// TIA Portal project "Project10" (V16)

(* hardware
DEVICE "GSD device_1"  GSD.Device.PN
   slot 0: "Rack"  Rack  V1.0
   slot 0: "SINAMICS-V90-PN"  SINAMICS V90 PN V1.0  6SL3 210-5Fxxx-xxFx  V1.00
      slot 0: "SINAMICS V90 PN V1.0"  SINAMICS V90 PN V1.0
      slot 1: "Drive_1"  Drive
         slot 0: "Module Access Point"  Module Access Point
         slot 1: "without PROFIsafe"  without PROFIsafe
      slot 1: "PN-IO"  PN-IO
         slot 1: "Port 1"  Port 1
         slot 2: "Port 2"  Port 2
   slot 2: "Standard telegram 3, PZD-5/9"  Standard telegram 3, PZD-5/9
DEVICE "S7-1200 station_1"  S7-1200 Station
   slot 0: "Rack_0"  S7-1200 Rack  Rack  V1.0
   slot 1: "PLC_1"  CPU 1214C AC/DC/Rly  6ES7 214-1BG40-0XB0  V4.3
*)

// ===== PLC "PLC_1"  CPU 1214C AC/DC/Rly =====

VAR_GLOBAL   // PLC tag table "Default tag table"
   "System_Byte" AT %MB1 : Byte;
   "FirstScan" AT %M1.0 : Bool;
   "DiagStatusUpdate" AT %M1.1 : Bool;
   "AlwaysTRUE" AT %M1.2 : Bool;
   "AlwaysFALSE" AT %M1.3 : Bool;
   "piston_ileri" AT %Q0.0 : Bool;
   "piston_geri" AT %Q0.1 : Bool;
   "pisron1_ilerde_sensörü" AT %I0.0 : Bool;
   "pisron1_geride_sensörü" AT %I0.1 : Bool;
   "pisron2_ilerde_sensörü" AT %I0.2 : Bool;
   "pisron2_geride_sensörü" AT %I0.3 : Bool;
   "hava_var_sinyal" AT %I0.7 : Bool;
   "acil_durum_basılı" AT %I0.4 : Bool;
   "otomatik_röle" AT %M2.0 : Bool;
   "manuel_röle" AT %M2.1 : Bool;
   "manuel_servo" AT %M2.2 : Bool;
   "manuel_piston" AT %M2.3 : Bool;
   "otomatik_hız1" AT %M2.4 : Bool;
   "otomatik_hız2" AT %M2.5 : Bool;
   "manuel_pistonlar_geri" AT %M2.6 : Bool;
   "manuel_pistonlar_ileri" AT %M2.7 : Bool;
   "oto_konum_1" AT %M3.0 : Bool;
   "oto_konum_2" AT %M3.1 : Bool;
   "oto_konum_3" AT %M3.2 : Bool;
   "oto_konum_4" AT %M3.3 : Bool;
   "oto_start" AT %M3.4 : Bool;
   "hız_bilgisi" AT %MD400 : Real;
   "konum_bilgisi" AT %MD450 : Real;
   "servo_on" AT %M12.0 : Bool;
   "servo_reset" AT %M12.1 : Bool;
   "pozisyon_start" AT %M12.2 : Bool;
   "pozisyon_tamamlandı" AT %M12.3 : Bool;
   "home_start" AT %M12.4 : Bool;
   "home_tamamlandı" AT %M12.5 : Bool;
   "Axis_1_Drive_IN" AT %I68.0 : "PD_TEL3_IN";
   "Axis_1_Drive_OUT" AT %Q64.0 : "PD_TEL3_OUT";
   "home_okey" AT %M12.6 : Bool;
   "pozi_okey" AT %M12.7 : Bool;
   "manuel_motor_ileri" AT %M13.0 : Bool;
   "manuel_motor_geri" AT %M13.1 : Bool;
   "oto_piston_ileri_start1" AT %M13.2 : Bool;
   "oto_piston_ileri_start2" AT %M13.3 : Bool;
   "oto_piston_ileri_start3" AT %M13.4 : Bool;
   "oto_piston_ileri_start4" AT %M13.5 : Bool;
   "oto_piston_geri_start1" AT %M13.6 : Bool;
   "oto_piston_geri_start2" AT %M13.7 : Bool;
   "oto_piston_geri_start3" AT %M14.0 : Bool;
   "oto_piston_geri_start4" AT %M14.1 : Bool;
   "sıra_izleme" AT %MW430 : Word;
   "oto_poz_start1" AT %M14.2 : Bool;
   "oto_poz_start2" AT %M14.3 : Bool;
   "oto_poz_start3" AT %M14.4 : Bool;
   "oto_poz_start4" AT %M14.5 : Bool;
   "oto_poz_start5" AT %M14.6 : Bool;
   "Tag_1" AT %M99.1 : Bool;
   "poz_set_düşür1" AT %M99.2 : Bool;
   "poz_set_düşür2" AT %M99.3 : Bool;
   "poz_set_düşür3" AT %M99.4 : Bool;
   "poz_set_düşür4" AT %M99.5 : Bool;
   "timer_set" AT %M99.6 : Bool;
   "Tag_2" AT %M98.0 : Bool;
   "timer_reset" AT %M98.1 : Bool;
   "servo_busy" AT %M98.2 : Bool;
   "hız1" AT %MD100 : Real;
   "arttırma" AT %M98.3 : Bool;
   "jog_meşgul" AT %M98.4 : Bool;
   "deneme" AT %M98.5 : Bool;
   "Clock_Byte" AT %MB0 : Byte;
   "Clock_10Hz" AT %M0.0 : Bool;
   "Clock_5Hz" AT %M0.1 : Bool;
   "Clock_2.5Hz" AT %M0.2 : Bool;
   "Clock_2Hz" AT %M0.3 : Bool;
   "Clock_1.25Hz" AT %M0.4 : Bool;
   "Clock_1Hz" AT %M0.5 : Bool;
   "Clock_0.625Hz" AT %M0.6 : Bool;
   "Clock_0.5Hz" AT %M0.7 : Bool;
   "COU_RST" AT %M3.5 : Bool;
   "DEN" AT %M3.6 : Bool;
END_VAR

DATA_BLOCK "DB_QR_DENEME"   // DB2
{ S7_Optimized_Access := 'FALSE' }
VERSION : 0.1
   VAR
      otomatik_manuel_mod_seçimi : Bool;
      manuel_seçim1 : Bool;
      manuel_seçim2 : Bool;
      manuel_piston_durum_oto_hız_bilgisi_1 : Bool;
      manuel_piston_durum_oto_hız_bilgisi_2 : Bool;
      oto_konum_bilgisi_1 : Bool;
      oto_konum_bilgisi_2 : Bool;
      oto_start : Bool;
      hız : Real;
      konum : Real;
      konum2 : Real;
      manuel_karşılaştır : Bool;
      sin : Bool;
      sinyal_oku2 : Bool;
      sinyal_oku : Bool;
   END_VAR
BEGIN
END_DATA_BLOCK

DATA_BLOCK "dbGenel"   // DB11
{ S7_Optimized_Access := 'TRUE' }
VERSION : 0.1
   VAR
      count : IEC_UCOUNTER;
   END_VAR
   VAR RETAIN
      Mikta : UInt;
   END_VAR
   VAR
      P_ken : Array[0..10] of Bool;
      reset : Bool;
      deneme : Bool;
      deneme_1 : Bool;
      deneme_2 : Bool;
   END_VAR
BEGIN
END_DATA_BLOCK

// folder: System blocks/Program resources

DATA_BLOCK "IEC_Timer_0_DB"   // DB8
{ S7_Optimized_Access := 'TRUE' }
AUTHOR : Simatic
FAMILY : IEC
NAME : IEC_TMR
VERSION : 1.0
// stored: InstanceOfName IEC_TIMER
"IEC_TIMER"
BEGIN
END_DATA_BLOCK

DATA_BLOCK "IEC_Timer_0_DB_1"   // DB9
{ S7_Optimized_Access := 'TRUE' }
AUTHOR : Simatic
FAMILY : IEC
NAME : IEC_TMR
VERSION : 1.0
// stored: InstanceOfName IEC_TIMER
"IEC_TIMER"
BEGIN
END_DATA_BLOCK

DATA_BLOCK "IEC_Timer_0_DB_2"   // DB10
{ S7_Optimized_Access := 'TRUE' }
AUTHOR : Simatic
FAMILY : IEC
NAME : IEC_TMR
VERSION : 1.0
// stored: InstanceOfName IEC_TIMER
"IEC_TIMER"
BEGIN
END_DATA_BLOCK

DATA_BLOCK "IEC_Timer_0_DB_5"   // DB13
{ S7_Optimized_Access := 'TRUE' }
AUTHOR : Simatic
FAMILY : IEC
NAME : IEC_TMR
VERSION : 1.0
// stored: InstanceOfName IEC_TIMER
"IEC_TIMER"
BEGIN
END_DATA_BLOCK

DATA_BLOCK "IEC_Counter_0_DB_1"   // DB14
{ S7_Optimized_Access := 'TRUE' }
AUTHOR : Simatic
FAMILY : IEC
NAME : CNTR
VERSION : 1.0
// stored: InstanceOfName IEC_COUNTER
"IEC_COUNTER"
BEGIN
END_DATA_BLOCK

// folder: (top level)

DATA_BLOCK "Axis_1"   // DB1, Motion_DB
{ S7_Optimized_Access := 'TRUE' }
AUTHOR : SIMATIC
FAMILY : BasicMC
NAME : TO_PosAx
VERSION : 6.0
// stored: InstanceOfName TO_PositioningAxis
"TO_PositioningAxis"
BEGIN
   // Axis.Encoder.TelegramAddressOutCU = %Q64.0
   // Axis.Encoder.TelegramAddressInCU = %I68.0
   // Axis.Encoder.DoNameCU = SINAMICS-V90-PN.Drive_1_Encoder1
   // Axis.Drive.TelegramAddressOutCU = %Q64.0
   // Axis.Drive.TelegramAddressInCU = %I68.0
   // Axis.Drive.TelegramType = 2
   // Axis.Drive.DoNameCU = SINAMICS-V90-PN.Drive_1
   // Axis.LengthUnitNormalized.Time = 1
   // Axis.LengthUnitNormalized.Distance = -2
   // Axis.Encoder.SelectedHscIndexCU = -1
   // Axis.Encoder.DbTypeCU = Classic
   // Axis.Drive.DbTypeCU = Classic
END_DATA_BLOCK

FUNCTION "fc_qr_eşleştir" : Void   // FC1, LAD
{ S7_Optimized_Access := 'TRUE' }
VERSION : 0.1
   VAR_TEMP   // added for the SCL form of the ladder/FBD networks
      _w1 : Bool;
   END_VAR
BEGIN

REGION Network 1: otomatik_manuel_mod_seçimi
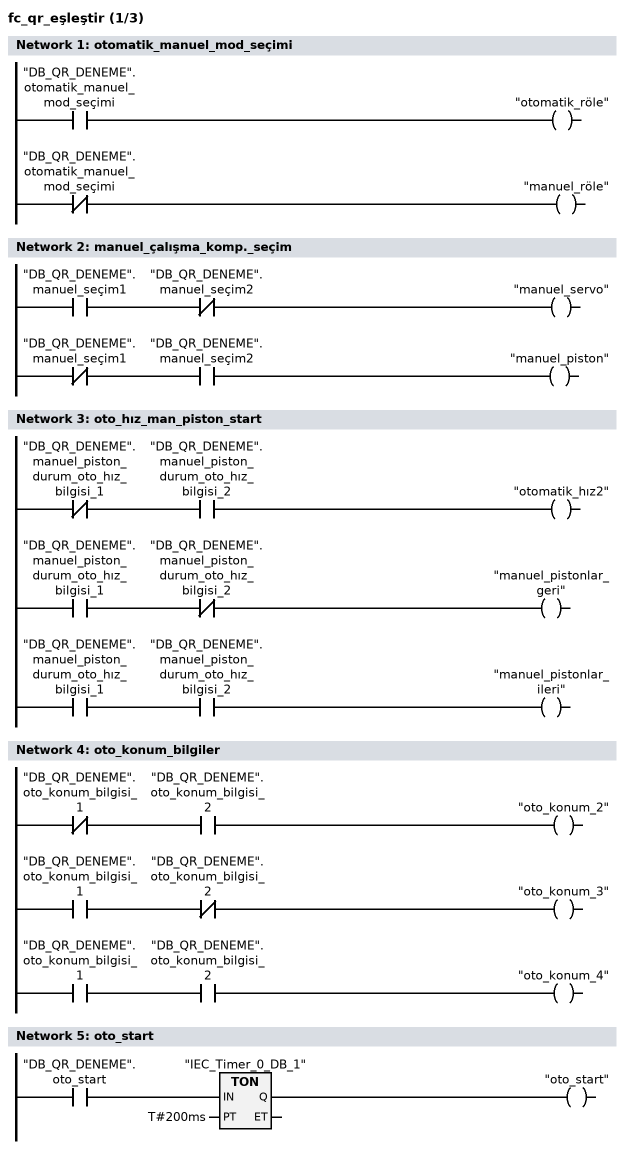
   RUNG wire#powerrail
      Contact( "DB_QR_DENEME".otomatik_manuel_mod_seçimi )
      Coil( "otomatik_röle" )
   END_RUNG
   RUNG wire#powerrail
      I_Contact( "DB_QR_DENEME".otomatik_manuel_mod_seçimi )
      Coil( "manuel_röle" )
   END_RUNG
   // the same network as SCL:
   "otomatik_röle" := "DB_QR_DENEME".otomatik_manuel_mod_seçimi;
   "manuel_röle" := NOT "DB_QR_DENEME".otomatik_manuel_mod_seçimi;
END_REGION

REGION Network 2: manuel_çalışma_komp._seçim
   RUNG wire#powerrail
      Contact( "DB_QR_DENEME".manuel_seçim1 )
      I_Contact( "DB_QR_DENEME".manuel_seçim2 )
      Coil( "manuel_servo" )
   END_RUNG
   RUNG wire#powerrail
      I_Contact( "DB_QR_DENEME".manuel_seçim1 )
      Contact( "DB_QR_DENEME".manuel_seçim2 )
      Coil( "manuel_piston" )
   END_RUNG
   // the same network as SCL:
   "manuel_servo" := "DB_QR_DENEME".manuel_seçim1 AND NOT "DB_QR_DENEME".manuel_seçim2;
   "manuel_piston" := NOT "DB_QR_DENEME".manuel_seçim1 AND "DB_QR_DENEME".manuel_seçim2;
END_REGION

REGION Network 3: oto_hız_man_piston_start
   RUNG wire#powerrail
      I_Contact( "DB_QR_DENEME".manuel_piston_durum_oto_hız_bilgisi_1 )
      Contact( "DB_QR_DENEME".manuel_piston_durum_oto_hız_bilgisi_2 )
      Coil( "otomatik_hız2" )
   END_RUNG
   RUNG wire#powerrail
      Contact( "DB_QR_DENEME".manuel_piston_durum_oto_hız_bilgisi_1 )
      I_Contact( "DB_QR_DENEME".manuel_piston_durum_oto_hız_bilgisi_2 )
      Coil( "manuel_pistonlar_geri" )
   END_RUNG
   RUNG wire#powerrail
      Contact( "DB_QR_DENEME".manuel_piston_durum_oto_hız_bilgisi_1 )
      Contact( "DB_QR_DENEME".manuel_piston_durum_oto_hız_bilgisi_2 )
      Coil( "manuel_pistonlar_ileri" )
   END_RUNG
   // the same network as SCL:
   "otomatik_hız2" := NOT "DB_QR_DENEME".manuel_piston_durum_oto_hız_bilgisi_1 AND "DB_QR_DENEME".manuel_piston_durum_oto_hız_bilgisi_2;
   "manuel_pistonlar_geri" := "DB_QR_DENEME".manuel_piston_durum_oto_hız_bilgisi_1 AND NOT "DB_QR_DENEME".manuel_piston_durum_oto_hız_bilgisi_2;
   "manuel_pistonlar_ileri" := "DB_QR_DENEME".manuel_piston_durum_oto_hız_bilgisi_1 AND "DB_QR_DENEME".manuel_piston_durum_oto_hız_bilgisi_2;
END_REGION

REGION Network 4: oto_konum_bilgiler
   RUNG wire#powerrail
      I_Contact( "DB_QR_DENEME".oto_konum_bilgisi_1 )
      Contact( "DB_QR_DENEME".oto_konum_bilgisi_2 )
      Coil( "oto_konum_2" )
   END_RUNG
   RUNG wire#powerrail
      Contact( "DB_QR_DENEME".oto_konum_bilgisi_1 )
      I_Contact( "DB_QR_DENEME".oto_konum_bilgisi_2 )
      Coil( "oto_konum_3" )
   END_RUNG
   RUNG wire#powerrail
      Contact( "DB_QR_DENEME".oto_konum_bilgisi_1 )
      Contact( "DB_QR_DENEME".oto_konum_bilgisi_2 )
      Coil( "oto_konum_4" )
   END_RUNG
   // the same network as SCL:
   "oto_konum_2" := NOT "DB_QR_DENEME".oto_konum_bilgisi_1 AND "DB_QR_DENEME".oto_konum_bilgisi_2;
   "oto_konum_3" := "DB_QR_DENEME".oto_konum_bilgisi_1 AND NOT "DB_QR_DENEME".oto_konum_bilgisi_2;
   "oto_konum_4" := "DB_QR_DENEME".oto_konum_bilgisi_1 AND "DB_QR_DENEME".oto_konum_bilgisi_2;
END_REGION

REGION Network 5: oto_start
   "IEC_Timer_0_DB_1".TON(IN := "DB_QR_DENEME".oto_start, PT := T#200ms);
   "oto_start" := "IEC_Timer_0_DB_1".Q;
END_REGION

REGION Network 6: hız_konum_atama
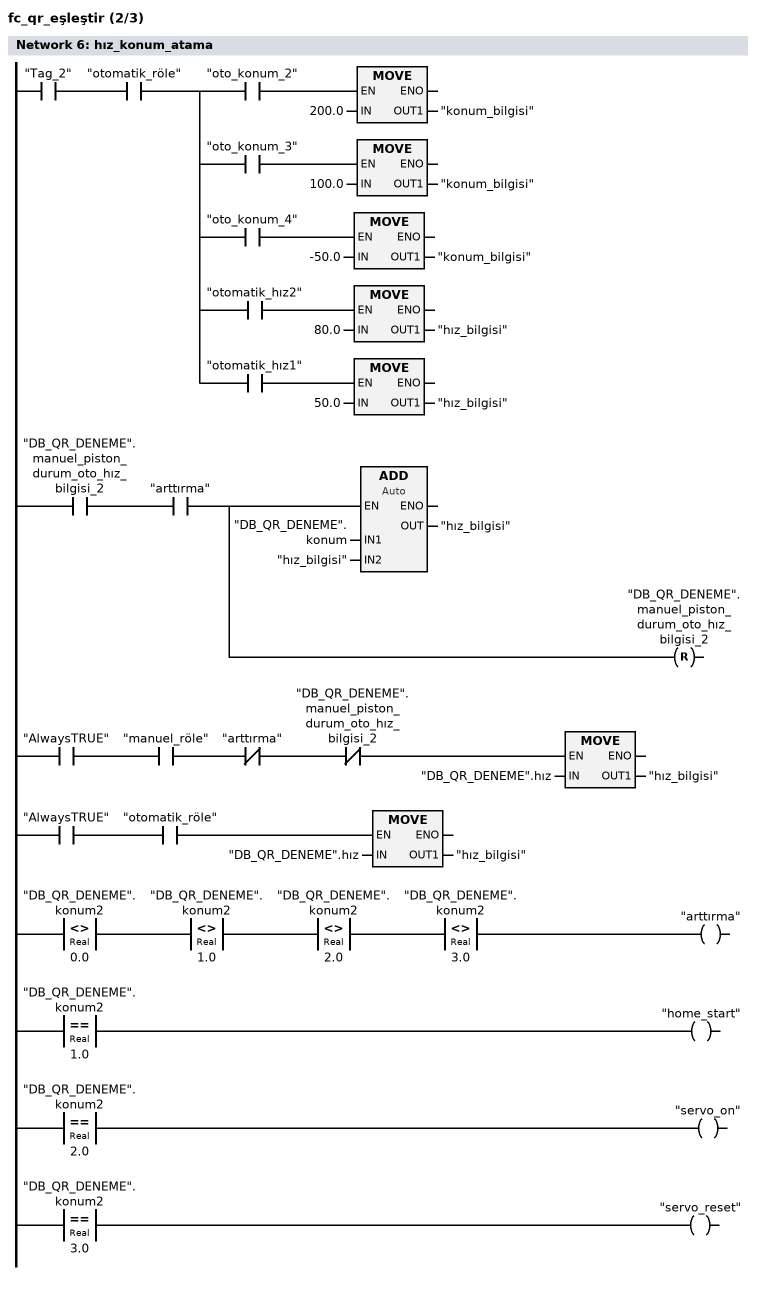
   RUNG wire#powerrail
      Contact( "Tag_2" )
      Contact( "otomatik_röle" )
      wire#w1
      Contact( "oto_konum_2" )
      Move(in := 200.0, out1 => "konum_bilgisi")
   END_RUNG
   RUNG wire#w1
      Contact( "oto_konum_3" )
      Move(in := 100.0, out1 => "konum_bilgisi")
   END_RUNG
   RUNG wire#w1
      Contact( "oto_konum_4" )
      Move(in := -50.0, out1 => "konum_bilgisi")
   END_RUNG
   RUNG wire#w1
      Contact( "otomatik_hız2" )
      Move(in := 80.0, out1 => "hız_bilgisi")
   END_RUNG
   RUNG wire#w1
      Contact( "otomatik_hız1" )
      Move(in := 50.0, out1 => "hız_bilgisi")
   END_RUNG
   RUNG wire#powerrail
      Contact( "DB_QR_DENEME".manuel_piston_durum_oto_hız_bilgisi_2 )
      Contact( "arttırma" )
      wire#w2
      Add(in1 := "DB_QR_DENEME".konum, in2 := "hız_bilgisi", out => "hız_bilgisi")
   END_RUNG
   RUNG wire#w2
      R_Coil( "DB_QR_DENEME".manuel_piston_durum_oto_hız_bilgisi_2 )
   END_RUNG
   RUNG wire#powerrail
      Contact( "AlwaysTRUE" )
      Contact( "manuel_röle" )
      I_Contact( "arttırma" )
      I_Contact( "DB_QR_DENEME".manuel_piston_durum_oto_hız_bilgisi_2 )
      Move(in := "DB_QR_DENEME".hız, out1 => "hız_bilgisi")
   END_RUNG
   RUNG wire#powerrail
      Contact( "AlwaysTRUE" )
      Contact( "otomatik_röle" )
      Move(in := "DB_QR_DENEME".hız, out1 => "hız_bilgisi")
   END_RUNG
   RUNG wire#powerrail
      { S7_Templates := "SrcType := Real" } NE_Contact(in1 := "DB_QR_DENEME".konum2, in2 := 0.0)
      { S7_Templates := "SrcType := Real" } NE_Contact(in1 := "DB_QR_DENEME".konum2, in2 := 1.0)
      { S7_Templates := "SrcType := Real" } NE_Contact(in1 := "DB_QR_DENEME".konum2, in2 := 2.0)
      { S7_Templates := "SrcType := Real" } NE_Contact(in1 := "DB_QR_DENEME".konum2, in2 := 3.0)
      Coil( "arttırma" )
   END_RUNG
   RUNG wire#powerrail
      { S7_Templates := "SrcType := Real" } EQ_Contact(in1 := "DB_QR_DENEME".konum2, in2 := 1.0)
      Coil( "home_start" )
   END_RUNG
   RUNG wire#powerrail
      { S7_Templates := "SrcType := Real" } EQ_Contact(in1 := "DB_QR_DENEME".konum2, in2 := 2.0)
      Coil( "servo_on" )
   END_RUNG
   RUNG wire#powerrail
      { S7_Templates := "SrcType := Real" } EQ_Contact(in1 := "DB_QR_DENEME".konum2, in2 := 3.0)
      Coil( "servo_reset" )
   END_RUNG
   // the same network as SCL:
   #_w1 := "Tag_2" AND "otomatik_röle";
   IF #_w1 AND "oto_konum_2" THEN "konum_bilgisi" := 200.0; END_IF;
   IF #_w1 AND "oto_konum_3" THEN "konum_bilgisi" := 100.0; END_IF;
   IF #_w1 AND "oto_konum_4" THEN "konum_bilgisi" := -50.0; END_IF;
   IF #_w1 AND "otomatik_hız2" THEN "hız_bilgisi" := 80.0; END_IF;
   IF #_w1 AND "otomatik_hız1" THEN "hız_bilgisi" := 50.0; END_IF;
   IF "DB_QR_DENEME".manuel_piston_durum_oto_hız_bilgisi_2 AND "arttırma" THEN
       "hız_bilgisi" := "DB_QR_DENEME".konum + "hız_bilgisi";
       "DB_QR_DENEME".manuel_piston_durum_oto_hız_bilgisi_2 := FALSE;
   END_IF;
   IF "AlwaysTRUE" AND "manuel_röle" AND NOT "arttırma" AND NOT "DB_QR_DENEME".manuel_piston_durum_oto_hız_bilgisi_2 THEN
       "hız_bilgisi" := "DB_QR_DENEME".hız;
   END_IF;
   IF "AlwaysTRUE" AND "otomatik_röle" THEN "hız_bilgisi" := "DB_QR_DENEME".hız; END_IF;
   "arttırma" := ("DB_QR_DENEME".konum2 <> 0.0) AND ("DB_QR_DENEME".konum2 <> 1.0) AND ("DB_QR_DENEME".konum2 <> 2.0) AND ("DB_QR_DENEME".konum2 <> 3.0);
   "home_start" := "DB_QR_DENEME".konum2 = 1.0;
   "servo_on" := "DB_QR_DENEME".konum2 = 2.0;
   "servo_reset" := "DB_QR_DENEME".konum2 = 3.0;
END_REGION

REGION Network 7
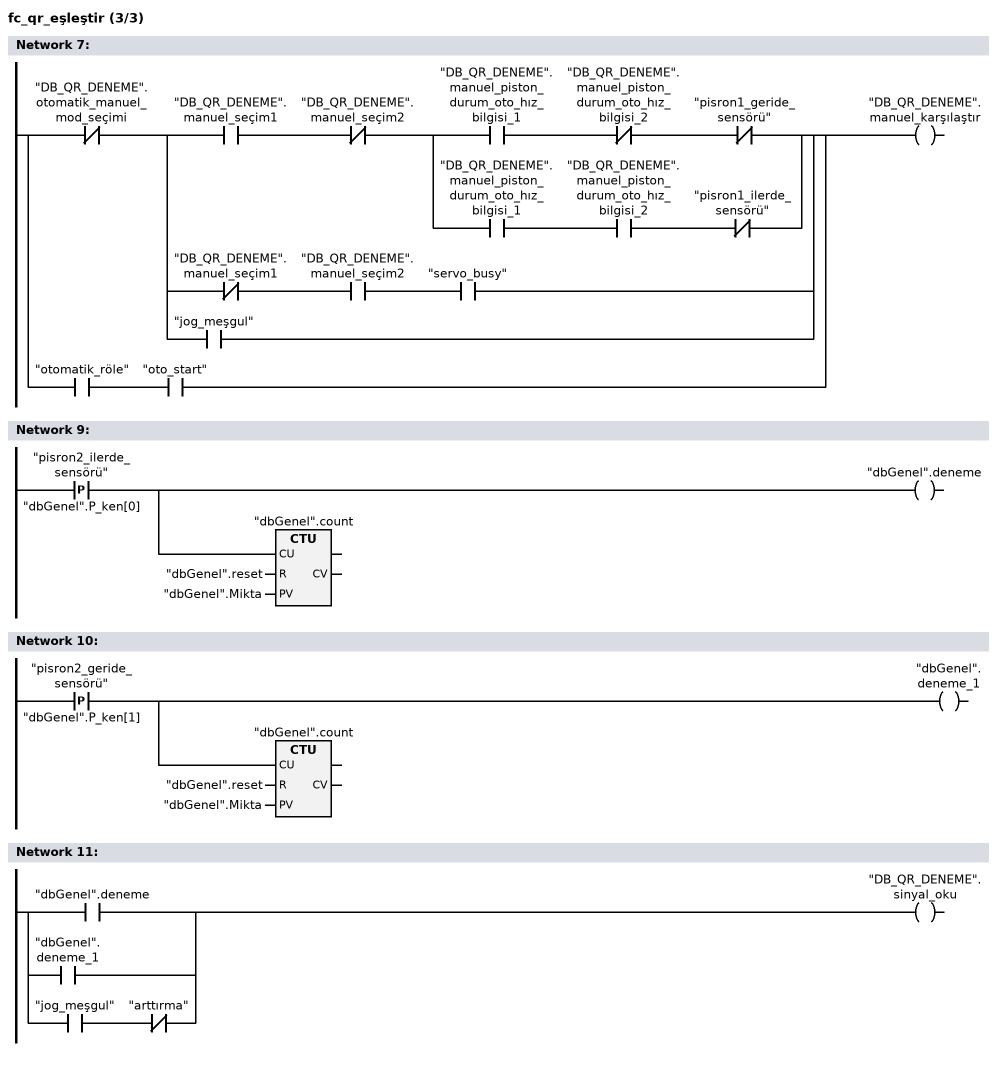
   RUNG wire#powerrail
      I_Contact( "DB_QR_DENEME".otomatik_manuel_mod_seçimi )
      wire#w1
      Contact( "DB_QR_DENEME".manuel_seçim1 )
      I_Contact( "DB_QR_DENEME".manuel_seçim2 )
      wire#w2
      Contact( "DB_QR_DENEME".manuel_piston_durum_oto_hız_bilgisi_1 )
      I_Contact( "DB_QR_DENEME".manuel_piston_durum_oto_hız_bilgisi_2 )
      I_Contact( "pisron1_geride_sensörü" )
      wire#w3
      Coil( "DB_QR_DENEME".manuel_karşılaştır )
   END_RUNG
   RUNG wire#w2
      Contact( "DB_QR_DENEME".manuel_piston_durum_oto_hız_bilgisi_1 )
      Contact( "DB_QR_DENEME".manuel_piston_durum_oto_hız_bilgisi_2 )
      I_Contact( "pisron1_ilerde_sensörü" )
   END_RUNG wire#w3
   RUNG wire#w1
      I_Contact( "DB_QR_DENEME".manuel_seçim1 )
      Contact( "DB_QR_DENEME".manuel_seçim2 )
      Contact( "servo_busy" )
   END_RUNG wire#w3
   RUNG wire#w1
      Contact( "jog_meşgul" )
   END_RUNG wire#w3
   RUNG wire#powerrail
      Contact( "otomatik_röle" )
      Contact( "oto_start" )
   END_RUNG wire#w3
   // the same network as SCL:
   "DB_QR_DENEME".manuel_karşılaştır := (NOT "DB_QR_DENEME".otomatik_manuel_mod_seçimi AND (("DB_QR_DENEME".manuel_seçim1 AND NOT "DB_QR_DENEME".manuel_seçim2 AND (("DB_QR_DENEME".manuel_piston_durum_oto_hız_bilgisi_1 AND NOT "DB_QR_DENEME".manuel_piston_durum_oto_hız_bilgisi_2 AND NOT "pisron1_geride_sensörü") OR ("DB_QR_DENEME".manuel_piston_durum_oto_hız_bilgisi_1 AND "DB_QR_DENEME".manuel_piston_durum_oto_hız_bilgisi_2 AND NOT "pisron1_ilerde_sensörü"))) OR (NOT "DB_QR_DENEME".manuel_seçim1 AND "DB_QR_DENEME".manuel_seçim2 AND "servo_busy") OR "jog_meşgul")) OR ("otomatik_röle" AND "oto_start");
END_REGION

REGION Network 9
   #_w1 := "pisron2_ilerde_sensörü" AND NOT "dbGenel".P_ken[0];   // rising edge of "pisron2_ilerde_sensörü"
   "dbGenel".P_ken[0] := "pisron2_ilerde_sensörü";
   "dbGenel".deneme := #_w1;
   "dbGenel".count.CTU(CU := #_w1, R := "dbGenel".reset, PV := "dbGenel".Mikta);
END_REGION

REGION Network 10
   #_w1 := "pisron2_geride_sensörü" AND NOT "dbGenel".P_ken[1];   // rising edge of "pisron2_geride_sensörü"
   "dbGenel".P_ken[1] := "pisron2_geride_sensörü";
   "dbGenel".deneme_1 := #_w1;
   "dbGenel".count.CTU(CU := #_w1, R := "dbGenel".reset, PV := "dbGenel".Mikta);
END_REGION

REGION Network 11
   RUNG wire#powerrail
      Contact( "dbGenel".deneme )
      wire#w1
      Coil( "DB_QR_DENEME".sinyal_oku )
   END_RUNG
   RUNG wire#powerrail
      Contact( "dbGenel".deneme_1 )
   END_RUNG wire#w1
   RUNG wire#powerrail
      Contact( "jog_meşgul" )
      I_Contact( "arttırma" )
   END_RUNG wire#w1
   // the same network as SCL:
   "DB_QR_DENEME".sinyal_oku := "dbGenel".deneme OR "dbGenel".deneme_1 OR ("jog_meşgul" AND NOT "arttırma");
END_REGION
END_FUNCTION

FUNCTION "fc_servo" : Void   // FC2, LAD
{ S7_Optimized_Access := 'TRUE' }
VERSION : 0.1
BEGIN

REGION Network 1
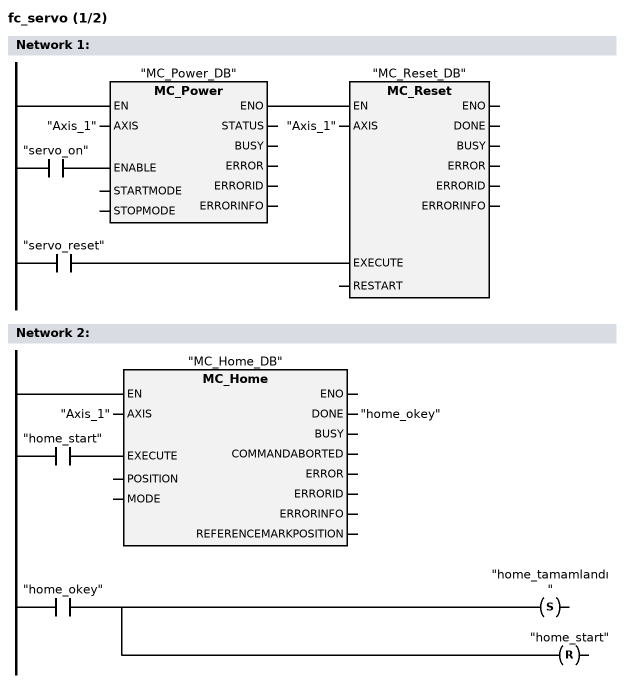
   // ENO of a box is taken as its EN; it also drops when the box reports an error
   "MC_Power_DB"(Axis := "Axis_1", Enable := "servo_on");   // MC_Power
   "MC_Reset_DB"(Axis := "Axis_1", Execute := "servo_reset");   // MC_Reset
END_REGION

REGION Network 2
   "MC_Home_DB"(Axis := "Axis_1", Execute := "home_start", Done => "home_okey");   // MC_Home
   IF "home_okey" THEN
       "home_tamamlandı" := TRUE;
       "home_start" := FALSE;
   END_IF;
END_REGION

REGION Network 3
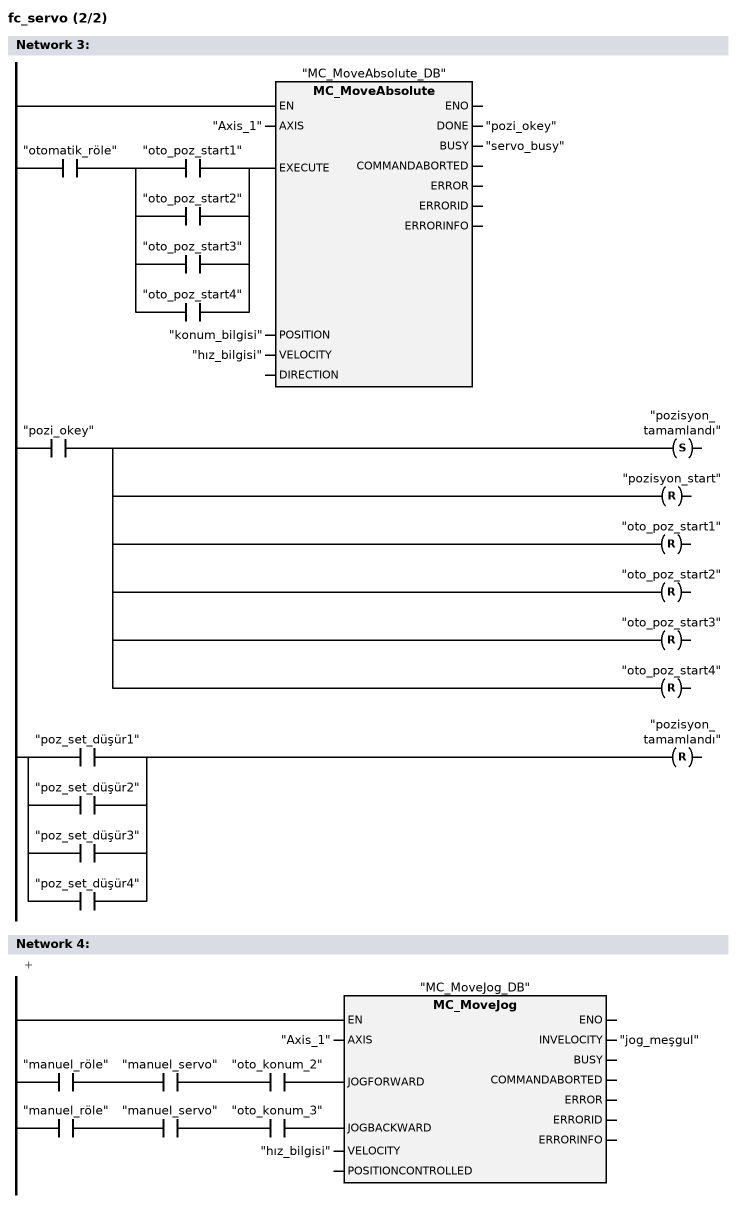
   "MC_MoveAbsolute_DB"(Axis := "Axis_1",   // MC_MoveAbsolute
                        Execute := "otomatik_röle" AND ("oto_poz_start1" OR "oto_poz_start2" OR "oto_poz_start3" OR "oto_poz_start4"),
                        Position := "konum_bilgisi",
                        Velocity := "hız_bilgisi",
                        Done => "pozi_okey",
                        Busy => "servo_busy");
   IF "pozi_okey" THEN
       "pozisyon_tamamlandı" := TRUE;
       "pozisyon_start" := FALSE;
       "oto_poz_start1" := FALSE;
       "oto_poz_start2" := FALSE;
       "oto_poz_start3" := FALSE;
       "oto_poz_start4" := FALSE;
   END_IF;
   IF "poz_set_düşür1" OR "poz_set_düşür2" OR "poz_set_düşür3" OR "poz_set_düşür4" THEN
       "pozisyon_tamamlandı" := FALSE;
   END_IF;
END_REGION

REGION Network 4
   // +
   "MC_MoveJog_DB"(Axis := "Axis_1",   // MC_MoveJog
                   JogForward := "manuel_röle" AND "manuel_servo" AND "oto_konum_2",
                   JogBackward := "manuel_röle" AND "manuel_servo" AND "oto_konum_3",
                   Velocity := "hız_bilgisi",
                   InVelocity => "jog_meşgul");
END_REGION
END_FUNCTION

FUNCTION "fc_piston" : Void   // FC3, LAD
{ S7_Optimized_Access := 'TRUE' }
VERSION : 0.1
   VAR_TEMP   // added for the SCL form of the ladder/FBD networks
      _w1 : Bool;
   END_VAR
BEGIN

REGION Network 1
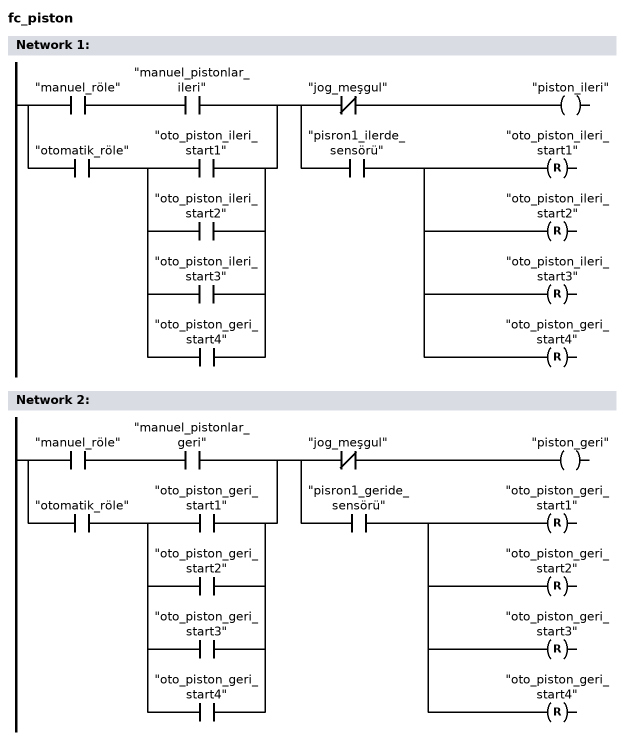
   RUNG wire#powerrail
      Contact( "manuel_röle" )
      Contact( "manuel_pistonlar_ileri" )
      wire#w1
      I_Contact( "jog_meşgul" )
      Coil( "piston_ileri" )
   END_RUNG
   RUNG wire#powerrail
      Contact( "otomatik_röle" )
      wire#w2
      Contact( "oto_piston_ileri_start1" )
   END_RUNG wire#w1
   RUNG wire#w2
      Contact( "oto_piston_ileri_start2" )
   END_RUNG wire#w1
   RUNG wire#w2
      Contact( "oto_piston_ileri_start3" )
   END_RUNG wire#w1
   RUNG wire#w2
      Contact( "oto_piston_geri_start4" )
   END_RUNG wire#w1
   RUNG wire#w1
      Contact( "pisron1_ilerde_sensörü" )
      wire#w3
      R_Coil( "oto_piston_ileri_start1" )
   END_RUNG
   RUNG wire#w3
      R_Coil( "oto_piston_ileri_start2" )
   END_RUNG
   RUNG wire#w3
      R_Coil( "oto_piston_ileri_start3" )
   END_RUNG
   RUNG wire#w3
      R_Coil( "oto_piston_geri_start4" )
   END_RUNG
   // the same network as SCL:
   #_w1 := ("manuel_röle" AND "manuel_pistonlar_ileri") OR ("otomatik_röle" AND ("oto_piston_ileri_start1" OR "oto_piston_ileri_start2" OR "oto_piston_ileri_start3" OR "oto_piston_geri_start4"));
   "piston_ileri" := #_w1 AND NOT "jog_meşgul";
   IF #_w1 AND "pisron1_ilerde_sensörü" THEN
       "oto_piston_ileri_start1" := FALSE;
       "oto_piston_ileri_start2" := FALSE;
       "oto_piston_ileri_start3" := FALSE;
       "oto_piston_geri_start4" := FALSE;
   END_IF;
END_REGION

REGION Network 2
   RUNG wire#powerrail
      Contact( "manuel_röle" )
      Contact( "manuel_pistonlar_geri" )
      wire#w1
      I_Contact( "jog_meşgul" )
      Coil( "piston_geri" )
   END_RUNG
   RUNG wire#powerrail
      Contact( "otomatik_röle" )
      wire#w2
      Contact( "oto_piston_geri_start1" )
   END_RUNG wire#w1
   RUNG wire#w2
      Contact( "oto_piston_geri_start2" )
   END_RUNG wire#w1
   RUNG wire#w2
      Contact( "oto_piston_geri_start3" )
   END_RUNG wire#w1
   RUNG wire#w2
      Contact( "oto_piston_geri_start4" )
   END_RUNG wire#w1
   RUNG wire#w1
      Contact( "pisron1_geride_sensörü" )
      wire#w3
      R_Coil( "oto_piston_geri_start1" )
   END_RUNG
   RUNG wire#w3
      R_Coil( "oto_piston_geri_start2" )
   END_RUNG
   RUNG wire#w3
      R_Coil( "oto_piston_geri_start3" )
   END_RUNG
   RUNG wire#w3
      R_Coil( "oto_piston_geri_start4" )
   END_RUNG
   // the same network as SCL:
   #_w1 := ("manuel_röle" AND "manuel_pistonlar_geri") OR ("otomatik_röle" AND ("oto_piston_geri_start1" OR "oto_piston_geri_start2" OR "oto_piston_geri_start3" OR "oto_piston_geri_start4"));
   "piston_geri" := #_w1 AND NOT "jog_meşgul";
   IF #_w1 AND "pisron1_geride_sensörü" THEN
       "oto_piston_geri_start1" := FALSE;
       "oto_piston_geri_start2" := FALSE;
       "oto_piston_geri_start3" := FALSE;
       "oto_piston_geri_start4" := FALSE;
   END_IF;
END_REGION
END_FUNCTION

FUNCTION "otomatik" : Void   // FC4, LAD
{ S7_Optimized_Access := 'TRUE' }
VERSION : 0.1
   VAR_TEMP   // added for the SCL form of the ladder/FBD networks
      _w1 : Bool;
      _w2 : Bool;
   END_VAR
BEGIN

REGION Network 1
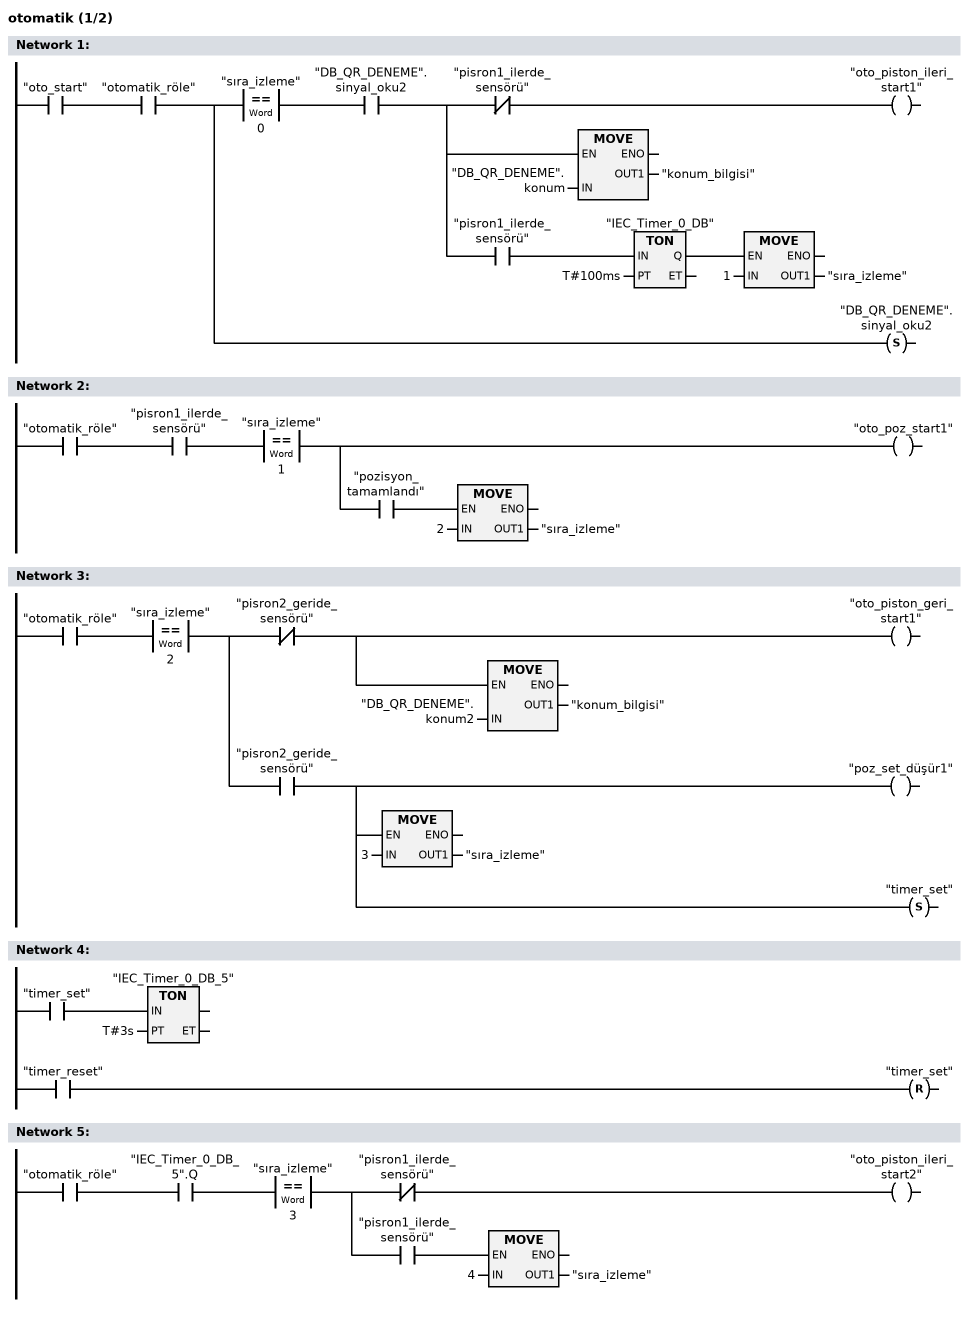
   #_w1 := "oto_start" AND "otomatik_röle";
   #_w2 := #_w1 AND ("sıra_izleme" = 0) AND "DB_QR_DENEME".sinyal_oku2;
   "oto_piston_ileri_start1" := #_w2 AND NOT "pisron1_ilerde_sensörü";
   IF #_w2 THEN "konum_bilgisi" := "DB_QR_DENEME".konum; END_IF;
   "IEC_Timer_0_DB".TON(IN := #_w2 AND "pisron1_ilerde_sensörü", PT := T#100ms);
   IF "IEC_Timer_0_DB".Q THEN "sıra_izleme" := 1; END_IF;
   IF #_w1 THEN "DB_QR_DENEME".sinyal_oku2 := TRUE; END_IF;
END_REGION

REGION Network 2
   RUNG wire#powerrail
      Contact( "otomatik_röle" )
      Contact( "pisron1_ilerde_sensörü" )
      { S7_Templates := "SrcType := Word" } EQ_Contact(in1 := "sıra_izleme", in2 := 1)
      wire#w1
      Coil( "oto_poz_start1" )
   END_RUNG
   RUNG wire#w1
      Contact( "pozisyon_tamamlandı" )
      Move(in := 2, out1 => "sıra_izleme")
   END_RUNG
   // the same network as SCL:
   "oto_poz_start1" := "otomatik_röle" AND "pisron1_ilerde_sensörü" AND ("sıra_izleme" = 1);
   IF "oto_poz_start1" AND "pozisyon_tamamlandı" THEN "sıra_izleme" := 2; END_IF;
END_REGION

REGION Network 3
   RUNG wire#powerrail
      Contact( "otomatik_röle" )
      { S7_Templates := "SrcType := Word" } EQ_Contact(in1 := "sıra_izleme", in2 := 2)
      wire#w1
      I_Contact( "pisron2_geride_sensörü" )
      wire#w2
      Coil( "oto_piston_geri_start1" )
   END_RUNG
   RUNG wire#w2
      Move(in := "DB_QR_DENEME".konum2, out1 => "konum_bilgisi")
   END_RUNG
   RUNG wire#w1
      Contact( "pisron2_geride_sensörü" )
      wire#w3
      Coil( "poz_set_düşür1" )
   END_RUNG
   RUNG wire#w3
      Move(in := 3, out1 => "sıra_izleme")
   END_RUNG
   RUNG wire#w3
      S_Coil( "timer_set" )
   END_RUNG
   // the same network as SCL:
   #_w1 := "otomatik_röle" AND ("sıra_izleme" = 2);
   "oto_piston_geri_start1" := #_w1 AND NOT "pisron2_geride_sensörü";
   IF "oto_piston_geri_start1" THEN "konum_bilgisi" := "DB_QR_DENEME".konum2; END_IF;
   "poz_set_düşür1" := #_w1 AND "pisron2_geride_sensörü";
   IF "poz_set_düşür1" THEN
       "sıra_izleme" := 3;
       "timer_set" := TRUE;
   END_IF;
END_REGION

REGION Network 4
   "IEC_Timer_0_DB_5".TON(IN := "timer_set", PT := T#3s);
   IF "timer_reset" THEN "timer_set" := FALSE; END_IF;
END_REGION

REGION Network 5
   RUNG wire#powerrail
      Contact( "otomatik_röle" )
      Contact( "IEC_Timer_0_DB_5".Q )
      { S7_Templates := "SrcType := Word" } EQ_Contact(in1 := "sıra_izleme", in2 := 3)
      wire#w1
      I_Contact( "pisron1_ilerde_sensörü" )
      Coil( "oto_piston_ileri_start2" )
   END_RUNG
   RUNG wire#w1
      Contact( "pisron1_ilerde_sensörü" )
      Move(in := 4, out1 => "sıra_izleme")
   END_RUNG
   // the same network as SCL:
   #_w1 := "otomatik_röle" AND "IEC_Timer_0_DB_5".Q AND ("sıra_izleme" = 3);
   "oto_piston_ileri_start2" := #_w1 AND NOT "pisron1_ilerde_sensörü";
   IF #_w1 AND "pisron1_ilerde_sensörü" THEN "sıra_izleme" := 4; END_IF;
END_REGION

REGION Network 6
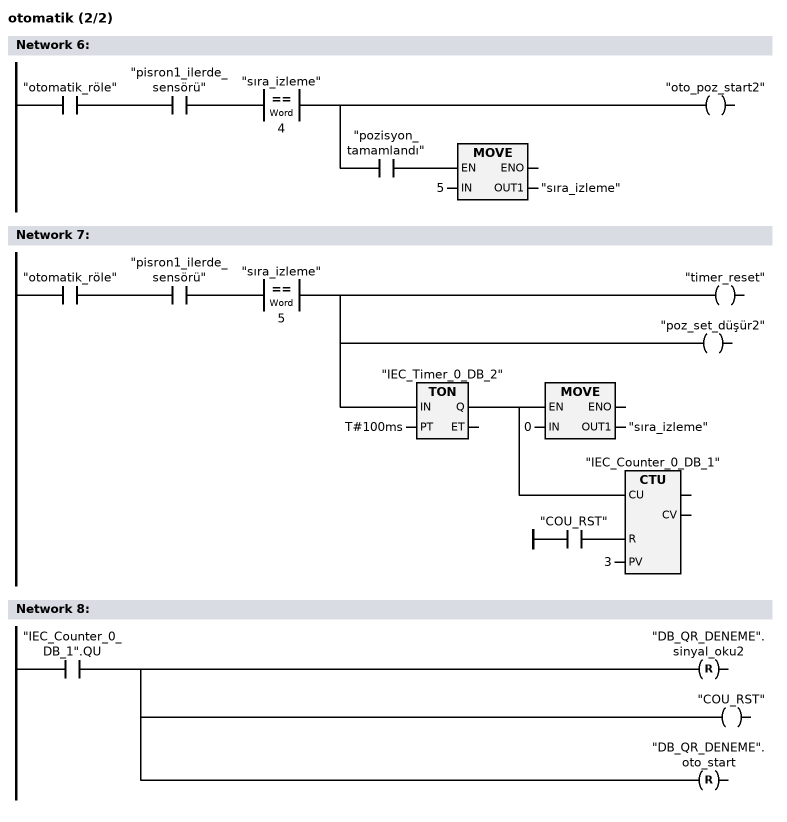
   RUNG wire#powerrail
      Contact( "otomatik_röle" )
      Contact( "pisron1_ilerde_sensörü" )
      { S7_Templates := "SrcType := Word" } EQ_Contact(in1 := "sıra_izleme", in2 := 4)
      wire#w1
      Coil( "oto_poz_start2" )
   END_RUNG
   RUNG wire#w1
      Contact( "pozisyon_tamamlandı" )
      Move(in := 5, out1 => "sıra_izleme")
   END_RUNG
   // the same network as SCL:
   "oto_poz_start2" := "otomatik_röle" AND "pisron1_ilerde_sensörü" AND ("sıra_izleme" = 4);
   IF "oto_poz_start2" AND "pozisyon_tamamlandı" THEN "sıra_izleme" := 5; END_IF;
END_REGION

REGION Network 7
   "timer_reset" := "otomatik_röle" AND "pisron1_ilerde_sensörü" AND ("sıra_izleme" = 5);
   "poz_set_düşür2" := "timer_reset";
   "IEC_Timer_0_DB_2".TON(IN := "timer_reset", PT := T#100ms);
   IF "IEC_Timer_0_DB_2".Q THEN "sıra_izleme" := 0; END_IF;
   "IEC_Counter_0_DB_1".CTU(CU := "IEC_Timer_0_DB_2".Q, R := "COU_RST", PV := 3);
END_REGION

REGION Network 8
   RUNG wire#powerrail
      Contact( "IEC_Counter_0_DB_1".QU )
      wire#w1
      R_Coil( "DB_QR_DENEME".sinyal_oku2 )
   END_RUNG
   RUNG wire#w1
      Coil( "COU_RST" )
   END_RUNG
   RUNG wire#w1
      R_Coil( "DB_QR_DENEME".oto_start )
   END_RUNG
   // the same network as SCL:
   IF "IEC_Counter_0_DB_1".QU THEN "DB_QR_DENEME".sinyal_oku2 := FALSE; END_IF;
   "COU_RST" := "IEC_Counter_0_DB_1".QU;
   IF "IEC_Counter_0_DB_1".QU THEN "DB_QR_DENEME".oto_start := FALSE; END_IF;
END_REGION
END_FUNCTION

ORGANIZATION_BLOCK "Main"   // OB1, LAD, ProgramCycle
TITLE = "Main Program Sweep (Cycle)"
{ S7_Optimized_Access := 'TRUE' }
VERSION : 0.1
   VAR_INPUT
      Initial_Call : Bool;   // Initial call of this OB
      Remanence : Bool;   // =True, if remanent data are available
   END_VAR
BEGIN

REGION Network 1
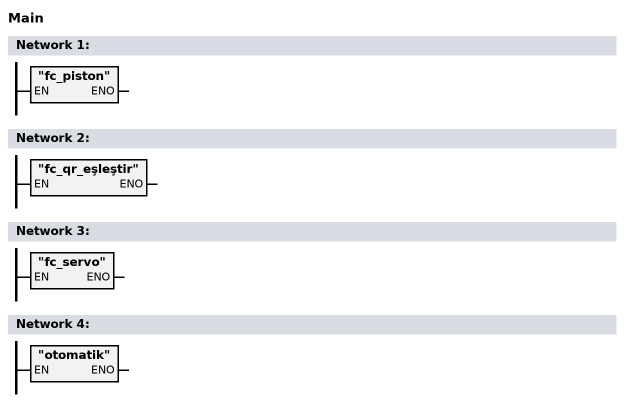
   RUNG wire#powerrail
      "fc_piston"()
   END_RUNG
   // the same network as SCL:
   "fc_piston"();
END_REGION

REGION Network 2
   RUNG wire#powerrail
      "fc_qr_eşleştir"()
   END_RUNG
   // the same network as SCL:
   "fc_qr_eşleştir"();
END_REGION

REGION Network 3
   RUNG wire#powerrail
      "fc_servo"()
   END_RUNG
   // the same network as SCL:
   "fc_servo"();
END_REGION

REGION Network 4
   RUNG wire#powerrail
      "otomatik"()
   END_RUNG
   // the same network as SCL:
   "otomatik"();
END_REGION
END_ORGANIZATION_BLOCK